FUNCTION_BLOCK FB_MQTTPublisher
VAR_INPUT
	(* published message *)
    Topic:			STRING(255) := 'RoboTel';
	Message:		STRING(255);
	Value:			STRING(255);
END_VAR
VAR_OUTPUT
	bPublished:		BOOL := TRUE;
END_VAR
VAR
	fbMqttClient:	FB_IotMqttClient;
    bSetParameter: 	BOOL := TRUE;
    sPayloadPub: 	STRING(255);
    bConnect:		BOOL := TRUE;
	bSubscribed:	BOOL;
    fbMessageQueue:	FB_IotMqttMessageQueue;
    //fbMessage      : FB_IotMqttMessage;
END_VAR

 IF bSetParameter THEN
    bSetParameter               := FALSE;
    fbMqttClient.sHostName      := 'primitivo.aip.de';
    fbMqttClient.nHostPort      := 1883;
    fbMqttClient.sClientId      := 'RoboTelPLC'; 
    fbMqttClient.sTopicPrefix   := ''; 
//  fbMqttClient.nKeepAlive     := 60; 
//  fbMqttClient.sUserName      := ;
//  fbMqttClient.sUserPassword  := ; 
//  fbMqttClient.stWill         := ; 
//  fbMqttClient.stTLS          := ;
    fbMqttClient.ipMessageQueue := fbMessageQueue;
END_IF

fbMqttClient.Execute(bConnect);

IF fbMqttClient.bConnected AND bPublished THEN
	sPayloadPub := CONCAT(Message, ' = ');
	sPayloadPub := CONCAT(sPayloadPub, Value);
	bPublished := fbMqttClient.Publish(	sTopic:= Topic, 
							pPayload:= ADR(sPayloadPub), 
							nPayloadSize:= LEN2(ADR(sPayloadPub))+0, // +1 just adds a \x0
							eQoS:= TcIotMqttQos.AtMostOnceDelivery, //TcIotMqttQos.AtMostOnceDelivery,  TcIotMqttQos.ExactlyOnceDelivery
							bRetain:= FALSE, 
							bQueue:= FALSE );
END_IF

END_FUNCTION_BLOCK

(* stored: Version 1.1.0.1, ProductVersion 3.1.4024.9
   POU FB_MQTTPublisher: Id {3d85d403-6f85-4edf-9b2a-1df91750ce4e}, SpecialFunc None *)
